INTERFACE I_Button

END_INTERFACE

(* stored: Version 1.1.0.1
   Itf I_Button: Id {d489b1a5-a2f1-4e4c-bd4f-d64b53deabd3} *)
